(* IEC 61131-3 sources: volt/packages/volt-lsp-iec/test-corpus/pro2193/Device/Plc Logic/Application/09 Misc/Library Manager/UDP, 19 files *)

(* ---- ERRORCODE.dut ---- *)
TYPE ERRORCODE :
(
	NO_ERROR,
	SOCKET_NONE_OPEN,
	SOCKET_NOTHING_RECEIVED,
	SOCKET_TIMEOUT,
	SOCKET_SELECT_FAILED,
	SOCKET_CREATE_FAILED,
	SOCKET_CLOSE_FAILED,
	INVALID_HANDLE,
	NO_DATA_AVAILABLE,
	WRONG_PARAMETER,
	IOCTL_FAILED,
	FD_SET_INIT_FAILED,
	SET_OPTION_BROADCAST_FAILED,
	SET_OPTION_MULTICAST_FAILED,
	SET_OPTION_ADD_MEMBERSHIP_FAILED,
	SET_OPTION_DROP_MEMBERSHIP_FAILED,
	BIND_FAILED,
	NOT_IMPLEMENTED
);
END_TYPE

(* ---- OS.dut ---- *)
TYPE OS :
(
	ANYSYSTEM := 0,
	LINUX
);
END_TYPE

(* ---- SOCK_RECV_MSG.dut ---- *)
TYPE SOCK_RECV_MSG :
STRUCT
	PBUFFER : POINTER TO BYTE;
	LENGTH : __XWORD;
	ADDRESS : SOCKADDRESS;
	MSGFLAGS : DWORD;
	MSGFLAGSSUPPORTED : DWORD;
END_STRUCT
END_TYPE

(* ---- SOCKETTYPE.dut ---- *)
TYPE SOCKETTYPE :
(
	UNICASTSOCKET := 0,
	BROADCASTSOCKET := 1,
	NETWORKBROADCASTSOCKET := 2,
	MULTICASTSOCKET := 3
);
END_TYPE

(* ---- CONSTANTS.gvl ---- *)
VAR_GLOBAL
	GC_FIRST_MULTICAST_IP : UDINT := 16#E0000000;
	GC_LAST_MULTICAST_IP : UDINT := 16#EFFFFFFF;
	GC_DEFAULT_SUBNETMASK : UDINT := 16#FFFFFF00;
END_VAR

(* ---- FD_CLR.pou ---- *)
FUNCTION FD_CLR : UDINT
VAR_INPUT
	HSOCKET : RTS_IEC_HANDLE;
	PFS : POINTER TO SysSocket.SOCKET_FD_SET;
END_VAR
END_FUNCTION

(* ---- IPARRAY_TO_IPSTRING.pou ---- *)
FUNCTION IPARRAY_TO_IPSTRING : STRING
VAR_INPUT
	ABYIPADDRESS : ARRAY [0..3] OF BYTE;
END_VAR
END_FUNCTION

(* ---- IPARRAY_TO_UDINT.pou ---- *)
FUNCTION IPARRAY_TO_UDINT : UDINT
VAR_INPUT
	ABYIPADDRESS : ARRAY [0..3] OF BYTE;
END_VAR
END_FUNCTION

(* ---- IPSTRING_TO_UDINT.pou ---- *)
FUNCTION IPSTRING_TO_UDINT : UDINT
VAR_INPUT
	SIPADDRESS : STRING;
END_VAR
END_FUNCTION

(* ---- IS_MULTICAST_GROUP.pou ---- *)
FUNCTION IS_MULTICAST_GROUP : BOOL
VAR_INPUT
	UDIIPADDRESS : UDINT;
END_VAR
END_FUNCTION

(* ---- MEMFORCESWAP.pou ---- *)
FUNCTION MEMFORCESWAP : INT
VAR_INPUT
	PBYBUFFER : POINTER TO BYTE;
	ISIZE : INT;
	ICOUNT : INT;
END_VAR
END_FUNCTION

(* ---- SWAP.pou ---- *)
FUNCTION SWAP : INT
VAR_INPUT
	PUC : POINTER TO BYTE;
	ISIZE : INT;
END_VAR
END_FUNCTION

(* ---- UDINT_TO_HEX.pou ---- *)
FUNCTION UDINT_TO_HEX : STRING(8)
VAR_INPUT
	VALUE : UDINT;
END_VAR
END_FUNCTION

(* ---- UDINT_TO_IPARRAY.pou ---- *)
FUNCTION UDINT_TO_IPARRAY : ARRAY [0..3] OF BYTE
VAR_INPUT
	UDIIPADDRESS : UDINT;
END_VAR
END_FUNCTION

(* ---- UDINT_TO_IPSTRING.pou ---- *)
FUNCTION UDINT_TO_IPSTRING : STRING
VAR_INPUT
	UDIIPADDRESS : UDINT;
END_VAR
END_FUNCTION

(* ---- UINT_TO_HEX.pou ---- *)
FUNCTION UINT_TO_HEX : STRING(4)
VAR_INPUT
	VALUE : UINT;
END_VAR
END_FUNCTION

(* ---- PERFORMANCEMONITOR.pou ---- *)
FUNCTION_BLOCK PERFORMANCEMONITOR
VAR_OUTPUT
	TMAXGAP : SYSTIME;
	TMINGAP : SYSTIME := 16#FFFFFFFF;
	TAVERAGEGAP : SYSTIME;
	TLASTGAP : SYSTIME;
	TTOTAL : SYSTIME;
END_VAR
VAR
	UDIDUMPCOUNT : UDINT;
	TLAST : SYSTIME;
	TSTART : SYSTIME;
	XSTARTED : BOOL;
END_VAR
END_FUNCTION_BLOCK

METHOD RESET
END_METHOD

METHOD START
END_METHOD

METHOD STOP
END_METHOD

(* ---- PORT.pou ---- *)
FUNCTION_BLOCK PORT
VAR
	_HSOCKET : SysTypes.RTS_IEC_HANDLE := SysTypes.HandleConstants.RTS_INVALID_HANDLE;
	_HBCSOCKET : SysTypes.RTS_IEC_HANDLE := SysTypes.HandleConstants.RTS_INVALID_HANDLE;
	_HNETWORKBCSOCKET : SysTypes.RTS_IEC_HANDLE := SysTypes.HandleConstants.RTS_INVALID_HANDLE;
	_HMULTICASTSOCKET : SysTypes.RTS_IEC_HANDLE := SysTypes.HandleConstants.RTS_INVALID_HANDLE;
	_XMULTICAST : BOOL;
	_UIRECVPORT : UINT;
	_UISENDPORT : UINT;
	_UDIIPADDRESS : UDINT;
	_SOCKETFDSET : SysSocket.SOCKET_FD_SET;
	_EOS : UDINT;
	_XOS_INITIALIZED : BOOL;
	_XNOBROADCASTSOCKET : BOOL;
	_REUSEADDRSOCKETOPTION : INT;
	_SYSSOCKSENDMONITOR : PerformanceMonitor;
	_SYSSOCKRECEIVEMONITOR : PerformanceMonitor;
	_SYSSOCKSELECTMONITOR : PerformanceMonitor;
	IPADDRESS : UDINT;
	OPERATINGSYSTEM : UDINT;
	RECEIVEPORT : UINT;
	REUSEADDRSOCKETOPTION : INT;
	SENDPORT : UINT;
	SOCKET : SysTypes.RTS_IEC_HANDLE;
END_VAR
END_FUNCTION_BLOCK

METHOD RECEIVE : SysTypes.RTS_IEC_RESULT
VAR_INPUT
	PBYDATA : POINTER TO BYTE;
	DIDATASIZE : __XINT;
END_VAR
VAR_OUTPUT
	UDIIPFROM : UDINT;
	UIPORTFROM : UINT;
	DIRECVSIZE : __XINT;
	ELOGCODE : ErrorCode;
END_VAR
END_METHOD

METHOD RECEIVE2 : SysTypes.RTS_IEC_RESULT
VAR_INPUT
	PBYDATA : POINTER TO BYTE;
	DIDATASIZE : __XINT;
END_VAR
VAR_OUTPUT
	UDIIPFROM : UDINT;
	UIPORTFROM : UINT;
	DIRECVSIZE : __XINT;
	ESOCKETTYPE : SocketType;
	ELOGCODE : ErrorCode;
END_VAR
END_METHOD

METHOD SEND : SysTypes.RTS_IEC_RESULT
VAR_INPUT
	UDIIPTO : UDINT;
	UIPORTTO : UINT;
	PBYDATA : POINTER TO BYTE;
	DIDATASIZE : __XINT;
END_VAR
VAR_OUTPUT
	DISENT : __XINT;
	ELOGCODE : ErrorCode;
END_VAR
END_METHOD

METHOD CLOSE : UDINT
END_METHOD

METHOD JOINGROUP : SysTypes.RTS_IEC_RESULT
VAR_INPUT
	UDIGROUPADDRESS : UDINT;
	UDIINTERFACEADDRESS : UDINT;
END_VAR
VAR_OUTPUT
	ELOGCODE : ErrorCode;
END_VAR
END_METHOD

METHOD LEAVEGROUP : SysTypes.RTS_IEC_RESULT
VAR_INPUT
	UDIGROUPADDRESS : UDINT;
	UDIINTERFACEADDRESS : UDINT;
END_VAR
VAR_OUTPUT
	ELOGCODE : ErrorCode;
END_VAR
END_METHOD

METHOD SETINTERFACE : SysTypes.RTS_IEC_RESULT
VAR_INPUT
	UDIIPADDRESS : UDINT;
END_VAR
VAR_OUTPUT
	ELOGCODE : ErrorCode;
END_VAR
END_METHOD

METHOD FB_EXIT : BOOL
VAR_INPUT
	BINCOPYCODE : BOOL;
END_VAR
END_METHOD

METHOD OPENRECVSOCKET : SysTypes.RTS_IEC_RESULT
VAR_OUTPUT
	ELOGCODE : ErrorCode;
END_VAR
END_METHOD

METHOD OPENSENDSOCKET : SysTypes.RTS_IEC_RESULT
VAR_OUTPUT
	ELOGCODE : ErrorCode;
END_VAR
END_METHOD

METHOD REOPEN : SysTypes.RTS_IEC_RESULT
VAR_OUTPUT
	ELOGCODE : ErrorCode;
END_VAR
END_METHOD

METHOD BIND : UDINT
VAR_INPUT
	UDIIPADDRESS : UDINT;
END_VAR
END_METHOD

METHOD FDISSET : BOOL
VAR_INPUT
	SOCKETFD_SET : SysSocket.SOCKET_FD_SET;
END_VAR
END_METHOD

METHOD FDSET
VAR_IN_OUT
	SOCKETFD_SET : SysSocket.SOCKET_FD_SET;
END_VAR
END_METHOD

METHOD GETOPTION : SysTypes.RTS_IEC_RESULT
VAR_INPUT
	DISOCKOPTION : DINT;
	PDIOPTION : POINTER TO DINT;
END_VAR
END_METHOD

METHOD IOCONTROL : SysTypes.RTS_IEC_RESULT
VAR_INPUT
	DICOMMAND : DINT;
	PDIPARAM : POINTER TO DINT;
END_VAR
END_METHOD

METHOD SETOPTION : SysTypes.RTS_IEC_RESULT
VAR_INPUT
	DISOCKOPTION : DINT;
	PDIOPTIONVALUE : POINTER TO DINT;
	DIOPTIONLENGTH : DINT;
END_VAR
END_METHOD

(* ---- UDPDRIVER.pou ---- *)
FUNCTION_BLOCK UDPDRIVER
VAR
	_SOCKETFDSET : SysSocket.SOCKET_FD_SET;
END_VAR
END_FUNCTION_BLOCK

METHOD BINDPORT : UDINT
VAR_INPUT
	PPORT : POINTER TO Port;
	UDILOCALIPADDRESS : UDINT;
END_VAR
VAR_OUTPUT
	ELOGCODE : ErrorCode;
END_VAR
END_METHOD

METHOD CLOSEPORT : SysTypes.RTS_IEC_RESULT
VAR_INPUT
	PPORT : POINTER TO Port;
END_VAR
VAR_OUTPUT
	ELOGCODE : ErrorCode;
END_VAR
END_METHOD

METHOD CREATEPORT : SysTypes.RTS_IEC_RESULT
VAR_INPUT
	PPORT : POINTER TO Port;
END_VAR
VAR_OUTPUT
	ELOGCODE : ErrorCode;
END_VAR
END_METHOD

METHOD CYCLICACTION : SysTypes.RTS_IEC_RESULT
END_METHOD

METHOD SELECT : SysTypes.RTS_IEC_RESULT
VAR_INPUT
	ITIMEOUT : INT;
END_VAR
VAR_OUTPUT
	DIREADY : DINT;
	ELOGCODE : ErrorCode;
END_VAR
VAR_IN_OUT
	STRRECVSET : SysSocket.SOCKET_FD_SET;
	STRSENDSET : SysSocket.SOCKET_FD_SET;
	STRERRORSET : SysSocket.SOCKET_FD_SET;
END_VAR
END_METHOD
